KUKA KRL program: ho_axor_atego.src, ho_axor_atego.dat

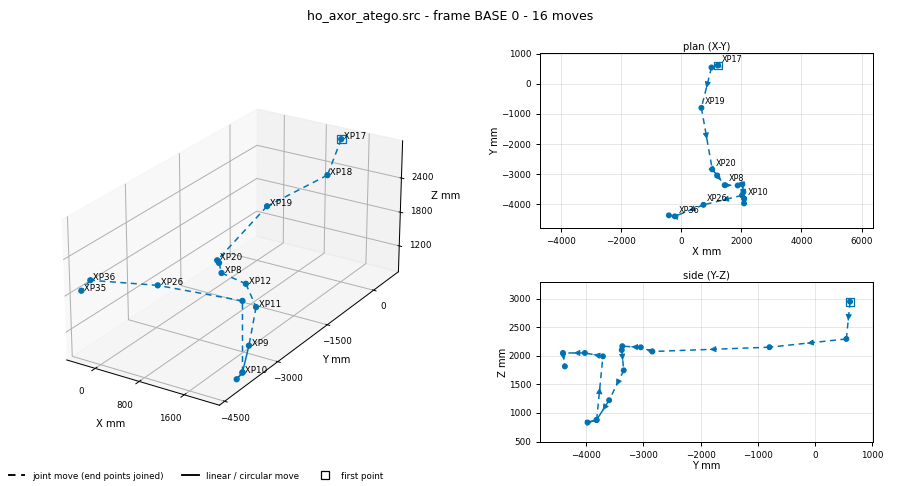
[picture p0: tool path of ho_axor_atego.src in frame BASE 0, 16 of 16 moves have a stored position in this frame; points joined in program order, loops and branches not executed]
--- ho_axor_atego.src ---
&ACCESS RVP
&REL 517
&COMMENT Pega Frente Axor_Atego
&PARAM DISKPATH = KRC:\R1\Program
&PARAM TEMPLATE = C:\KRC\Roboter\Template\vorgabe
&PARAM EDITMASK = *
DEF ho_axor_atego( )
;FOLD INI
  ;FOLD BASISTECH INI
    GLOBAL INTERRUPT DECL 3 WHEN $STOPMESS==TRUE DO IR_STOPM ( )
    INTERRUPT ON 3
    BAS (#INITMOV,0 )
  ;ENDFOLD (BASISTECH INI)
;FOLD SPOTTECH INI
USERSPOT(#INIT)
;ENDFOLD (SPOTTECH INI)
;FOLD GRIPPERTECH INI
USER_GRP(0,DUMMY,DUMMY,GDEFAULT)
;ENDFOLD (GRIPPERTECH INI)
  ;FOLD USER INI
    ;Make your modifications here

  ;ENDFOLD (USER INI)
;ENDFOLD (INI)

; Caracterização dos meios de produção:
; Changes: Pega Frontal Axor/Atego
; Versão Atual:11/08/2015
; Name: P13.050-R4

chk_w6_wechs_ok ( )  ; CHECK TOOL: GRIPPER AXOR

;FOLD PTP P17 Vel=100 % PDAT16 Tool[6]:GARRA AXOR Base[0];%{PE}%R 8.2.20,%MKUKATPBASIS,%CMOVE,%VPTP,%P 1:PTP, 2:P17, 3:, 5:100, 7:PDAT16
$BWDSTART=FALSE
PDAT_ACT=PPDAT16
FDAT_ACT=FP17
BAS(#PTP_PARAMS,100)
PTP XP17
;ENDFOLD

;FOLD PTP P18 CONT Vel=100 % PDAT17 Tool[6]:GARRA AXOR Base[0];%{PE}%R 8.2.20,%MKUKATPBASIS,%CMOVE,%VPTP,%P 1:PTP, 2:P18, 3:C_DIS, 5:100, 7:PDAT17
$BWDSTART=FALSE
PDAT_ACT=PPDAT17
FDAT_ACT=FP18
BAS(#PTP_PARAMS,100)
PTP XP18 C_DIS
;ENDFOLD
;FOLD PTP P19 CONT Vel=100 % PDAT18 Tool[6]:GARRA AXOR Base[0];%{PE}%R 8.2.20,%MKUKATPBASIS,%CMOVE,%VPTP,%P 1:PTP, 2:P19, 3:C_DIS, 5:100, 7:PDAT18
$BWDSTART=FALSE
PDAT_ACT=PPDAT18
FDAT_ACT=FP19
BAS(#PTP_PARAMS,100)
PTP XP19 C_DIS
;ENDFOLD

;FOLD ; LIBERACAO P/ RETIRAR PECA NO DISPOSITIVO;%{PE}%R 8.2.20,%MKUKATPBASIS,%CCOMMENT,%VNORMAL,%P 2:LIBERACAO  P/  RETIRAR  PECA  NO  DISPOSITIVO
;ENDFOLD
;FOLD PTP P20 CONT Vel=100 % PDAT19 Tool[6]:GARRA AXOR Base[0];%{PE}%R 8.2.20,%MKUKATPBASIS,%CMOVE,%VPTP,%P 1:PTP, 2:P20, 3:C_DIS, 5:100, 7:PDAT19
$BWDSTART=FALSE
PDAT_ACT=PPDAT19
FDAT_ACT=FP20
BAS(#PTP_PARAMS,100)
PTP XP20 C_DIS
;ENDFOLD

;FOLD OUT 3352 'R4 busca peca Actros' State=TRUE ;%{PE}%R 8.2.20,%MKUKATPBASIS,%COUT,%VOUTX,%P 2:3352, 3:R4 busca peca Actros, 5:TRUE, 6:
$OUT[3352]=TRUE
;ENDFOLD
;FOLD WAIT FOR ( IN 3352 'Aguarda lib buscar peca Actros' );%{PE}%R 8.2.20,%MKUKATPBASIS,%CEXT_WAIT_FOR,%VEXT_WAIT_FOR,%P 2:, 4:, 5:$IN, 6:3352, 7:Aguarda lib buscar peca Actros, 9:
WAIT FOR  ( $IN[3352] )
;ENDFOLD
;FOLD OUT 3352 'R4 busca peca Actros' State=FALSE ;%{PE}%R 8.2.20,%MKUKATPBASIS,%COUT,%VOUTX,%P 2:3352, 3:R4 busca peca Actros, 5:FALSE, 6:
$OUT[3352]=FALSE
;ENDFOLD
;FOLD OUT 3342 'Fora area externa' State=FALSE ;%{PE}%R 8.2.20,%MKUKATPBASIS,%COUT,%VOUTX,%P 2:3342, 3:Fora area externa, 5:FALSE, 6:
$OUT[3342]=FALSE
;ENDFOLD

;FOLD PTP P15 CONT Vel=100 % PDAT14 Tool[6]:GARRA AXOR Base[0];%{PE}%R 8.2.20,%MKUKATPBASIS,%CMOVE,%VPTP,%P 1:PTP, 2:P15, 3:C_DIS, 5:100, 7:PDAT14
$BWDSTART=FALSE
PDAT_ACT=PPDAT14
FDAT_ACT=FP15
BAS(#PTP_PARAMS,100)
PTP XP15 C_DIS
;ENDFOLD
;FOLD PTP P8 CONT Vel=100 % PDAT9 Tool[6]:GARRA AXOR Base[0];%{PE}%R 8.2.20,%MKUKATPBASIS,%CMOVE,%VPTP,%P 1:PTP, 2:P8, 3:C_DIS, 5:100, 7:PDAT9
$BWDSTART=FALSE
PDAT_ACT=PPDAT9
FDAT_ACT=FP8
BAS(#PTP_PARAMS,100)
PTP XP8 C_DIS
;ENDFOLD
;FOLD PTP P12 CONT Vel=100 % PDAT12 Tool[6]:GARRA AXOR Base[0];%{PE}%R 8.2.20,%MKUKATPBASIS,%CMOVE,%VPTP,%P 1:PTP, 2:P12, 3:C_DIS, 5:100, 7:PDAT12
$BWDSTART=FALSE
PDAT_ACT=PPDAT12
FDAT_ACT=FP12
BAS(#PTP_PARAMS,100)
PTP XP12 C_DIS
;ENDFOLD
;FOLD PTP P11 CONT Vel=100 % PDAT11 Tool[6]:GARRA AXOR Base[0];%{PE}%R 8.2.20,%MKUKATPBASIS,%CMOVE,%VPTP,%P 1:PTP, 2:P11, 3:C_DIS, 5:100, 7:PDAT11
$BWDSTART=FALSE
PDAT_ACT=PPDAT11
FDAT_ACT=FP11
BAS(#PTP_PARAMS,100)
PTP XP11 C_DIS
;ENDFOLD
;FOLD PTP P9 CONT Vel=100 % PDAT10 Tool[6]:GARRA AXOR Base[0];%{PE}%R 8.2.20,%MKUKATPBASIS,%CMOVE,%VPTP,%P 1:PTP, 2:P9, 3:C_DIS, 5:100, 7:PDAT10
$BWDSTART=FALSE
PDAT_ACT=PPDAT10
FDAT_ACT=FP9
BAS(#PTP_PARAMS,100)
PTP XP9 C_DIS
;ENDFOLD

;FOLD SET Z1.1/Z1.2/Z1.3 AXOR State=OPN GDAT12;%{PE}%R 8.2.1,%MKUKATPGRP,%CGRP,%VGRP,%P 2:5, 4:1, 5:#NO, 6:GDAT12, 8:0, 10:0
H50(GRP,5,1,GGDAT12)
;ENDFOLD
;FOLD SET Z2.1/Z2.2 AXOR State=OPN GDAT13;%{PE}%R 8.2.1,%MKUKATPGRP,%CGRP,%VGRP,%P 2:6, 4:1, 5:#NO, 6:GDAT13, 8:0, 10:0
H50(GRP,6,1,GGDAT13)
;ENDFOLD
;FOLD SET Z3.1/Z3.2 AXOR State=OPN GDAT14;%{PE}%R 8.2.1,%MKUKATPGRP,%CGRP,%VGRP,%P 2:7, 4:1, 5:#NO, 6:GDAT14, 8:0, 10:0
H50(GRP,7,1,GGDAT14)
;ENDFOLD
chk_w6_grp1_opn ()
chk_w6_grp2_opn ()
chk_w6_grp3_opn ()

;FOLD LIN P10 CONT Vel=0.5 m/s CPDAT3 Tool[6]:GARRA AXOR Base[0];%{PE}%R 8.2.20,%MKUKATPBASIS,%CMOVE,%VLIN,%P 1:LIN, 2:P10, 3:C_DIS C_DIS, 5:0.5, 7:CPDAT3
$BWDSTART=FALSE
LDAT_ACT=LCPDAT3
FDAT_ACT=FP10
BAS(#CP_PARAMS,0.5)
LIN XP10 C_DIS C_DIS
;ENDFOLD

;FOLD ; POSICAO DE PEGA DA PECA;%{PE}%R 8.2.20,%MKUKATPBASIS,%CCOMMENT,%VNORMAL,%P 2:POSICAO  DE  PEGA  DA  PECA
;ENDFOLD
;FOLD LIN P14 CONT Vel=0.5 m/s CPDAT4 Tool[6]:GARRA AXOR Base[0];%{PE}%R 8.2.20,%MKUKATPBASIS,%CMOVE,%VLIN,%P 1:LIN, 2:P14, 3:C_DIS C_DIS, 5:0.5, 7:CPDAT4
$BWDSTART=FALSE
LDAT_ACT=LCPDAT4
FDAT_ACT=FP14
BAS(#CP_PARAMS,0.5)
LIN XP14 C_DIS C_DIS
;ENDFOLD

IF (NOT(GHOST())) THEN
;FOLD WAIT FOR ( IN 489 'Presença de peça 1 - Axor' AND IN 490 'Presença de peça 2 - Axor' );%{PE}%R 8.2.20,%MKUKATPBASIS,%CEXT_WAIT_FOR,%VEXT_WAIT_FOR,%P 2:, 4:, 5:$IN, 6:489, 7:Presença de peça 1 - Axor, 8:AND, 9:, 10:$IN, 11:490, 12:Presença de peça 2 - Axor, 14:
WAIT FOR  ( $IN[489] AND $IN[490] )
;ENDFOLD
ENDIF

;FOLD SET Z1.1/Z1.2/Z1.3 AXOR State=CLO GDAT9;%{PE}%R 8.2.1,%MKUKATPGRP,%CGRP,%VGRP,%P 2:5, 4:2, 5:#NO, 6:GDAT9, 8:0, 10:0
H50(GRP,5,2,GGDAT9)
;ENDFOLD
;FOLD SET Z2.1/Z2.2 AXOR State=CLO GDAT10;%{PE}%R 8.2.1,%MKUKATPGRP,%CGRP,%VGRP,%P 2:6, 4:2, 5:#NO, 6:GDAT10, 8:0, 10:0
H50(GRP,6,2,GGDAT10)
;ENDFOLD
;FOLD SET Z3.1/Z3.2 AXOR State=CLO GDAT11;%{PE}%R 8.2.1,%MKUKATPGRP,%CGRP,%VGRP,%P 2:7, 4:2, 5:#NO, 6:GDAT11, 8:0, 10:0
H50(GRP,7,2,GGDAT11)
;ENDFOLD
chk_w6_grp1_clo ()
chk_w6_grp2_clo ()
chk_w6_grp3_clo ()

;FOLD OUT 3349 'R4 pegou peca' State=TRUE ;%{PE}%R 8.2.20,%MKUKATPBASIS,%COUT,%VOUTX,%P 2:3349, 3:R4 pegou peca, 5:TRUE, 6:
$OUT[3349]=TRUE
;ENDFOLD
;FOLD OUT 3350 'R4 solicita lib sair magazine' State=TRUE ;%{PE}%R 8.2.20,%MKUKATPBASIS,%COUT,%VOUTX,%P 2:3350, 3:R4 solicita lib sair magazine, 5:TRUE, 6:
$OUT[3350]=TRUE
;ENDFOLD
;FOLD WAIT FOR ( IN 3349 'Aguarda lib sair magazine' );%{PE}%R 8.2.20,%MKUKATPBASIS,%CEXT_WAIT_FOR,%VEXT_WAIT_FOR,%P 2:, 4:, 5:$IN, 6:3349, 7:Aguarda lib sair magazine, 9:
WAIT FOR  ( $IN[3349] )
;ENDFOLD
;FOLD OUT 3350 'R4 solicita lib sair magazine' State=FALSE ;%{PE}%R 8.2.20,%MKUKATPBASIS,%COUT,%VOUTX,%P 2:3350, 3:R4 solicita lib sair magazine, 5:FALSE, 6:
$OUT[3350]=FALSE
;ENDFOLD

;FOLD LIN P22 CONT Vel=0.1 m/s CPDAT6 Tool[6]:GARRA AXOR Base[0];%{PE}%R 8.2.20,%MKUKATPBASIS,%CMOVE,%VLIN,%P 1:LIN, 2:P22, 3:C_DIS C_DIS, 5:0.1, 7:CPDAT6
$BWDSTART=FALSE
LDAT_ACT=LCPDAT6
FDAT_ACT=FP22
BAS(#CP_PARAMS,0.1)
LIN XP22 C_DIS C_DIS
;ENDFOLD

IF (NOT(GHOST())) THEN
;FOLD WAIT FOR ( IN 489 'Presença de peça 1 - Axor' AND IN 490 'Presença de peça 2 - Axor' );%{PE}%R 8.2.20,%MKUKATPBASIS,%CEXT_WAIT_FOR,%VEXT_WAIT_FOR,%P 2:, 4:, 5:$IN, 6:489, 7:Presença de peça 1 - Axor, 8:AND, 9:, 10:$IN, 11:490, 12:Presença de peça 2 - Axor, 14:
WAIT FOR  ( $IN[489] AND $IN[490] )
;ENDFOLD
ENDIF

;FOLD PTP P25 CONT Vel=100 % PDAT23 Tool[6]:GARRA AXOR Base[0];%{PE}%R 8.2.20,%MKUKATPBASIS,%CMOVE,%VPTP,%P 1:PTP, 2:P25, 3:C_DIS, 5:100, 7:PDAT23
$BWDSTART=FALSE
PDAT_ACT=PPDAT23
FDAT_ACT=FP25
BAS(#PTP_PARAMS,100)
PTP XP25 C_DIS
;ENDFOLD
;FOLD PTP P26 CONT Vel=100 % PDAT24 Tool[6]:GARRA AXOR Base[0];%{PE}%R 8.2.20,%MKUKATPBASIS,%CMOVE,%VPTP,%P 1:PTP, 2:P26, 3:C_DIS, 5:100, 7:PDAT24
$BWDSTART=FALSE
PDAT_ACT=PPDAT24
FDAT_ACT=FP26
BAS(#PTP_PARAMS,100)
PTP XP26 C_DIS
;ENDFOLD
;FOLD PTP P36 CONT Vel=100 % PDAT33 Tool[6]:GARRA AXOR Base[0];%{PE}%R 8.2.20,%MKUKATPBASIS,%CMOVE,%VPTP,%P 1:PTP, 2:P36, 3:C_DIS, 5:100, 7:PDAT33
$BWDSTART=FALSE
PDAT_ACT=PPDAT33
FDAT_ACT=FP36
BAS(#PTP_PARAMS,100)
PTP XP36 C_DIS
;ENDFOLD
;FOLD PTP P35 CONT Vel=100 % PDAT32 Tool[6]:GARRA AXOR Base[0];%{PE}%R 8.2.20,%MKUKATPBASIS,%CMOVE,%VPTP,%P 1:PTP, 2:P35, 3:C_DIS, 5:100, 7:PDAT32
$BWDSTART=FALSE
PDAT_ACT=PPDAT32
FDAT_ACT=FP35
BAS(#PTP_PARAMS,100)
PTP XP35 C_DIS
;ENDFOLD

END

--- ho_axor_atego.dat ---
&ACCESS RVP
&REL 517
&COMMENT Pega Frente Axor_Atego
&PARAM DISKPATH = KRC:\R1\Program
&PARAM TEMPLATE = C:\KRC\Roboter\Template\vorgabe
&PARAM EDITMASK = *
DEFDAT  ho_axor_atego
;FOLD EXTERNAL DECLARATIONS;%{PE}%MKUKATPBASIS,%CEXT,%VCOMMON,%P
;FOLD GRIPPERTECH EXT
EXT  H50 (INT  :IN,INT  :IN,INT  :IN,GRP_TYP  :IN )
;ENDFOLD (GRIPPERTECH EXT)
;FOLD SPOTTECH EXT
EXT  USERSPOT (S_COMMAND  :IN,SPOT_TYPE  :IN )
;ENDFOLD (SPOTTECH EXT)
;FOLD BASISTECH EXT;%{PE}%MKUKATPBASIS,%CEXT,%VEXT,%P
EXT  BAS (BAS_COMMAND  :IN,REAL  :IN )
DECL INT SUCCESS
;ENDFOLD (BASISTECH EXT)
;FOLD USER EXT;%{E}%MKUKATPUSER,%CEXT,%VEXT,%P
;Make your modifications here

;ENDFOLD (USER EXT)
;ENDFOLD (EXTERNAL DECLARATIONS)
DECL BASIS_SUGG_T LAST_BASIS={POINT1[] "P37                     ",POINT2[] "P37                     ",CP_PARAMS[] "CPDAT7                  ",PTP_PARAMS[] "PDAT34                  ",CONT[] "C_DIS                   ",CP_VEL[] "0.1                     ",PTP_VEL[] "100                     ",SYNC_PARAMS[] "SYNCDAT                 ",SPL_NAME[] "S0                      "}
DECL E6POS XP8={X 1445.68298,Y -3370.3269,Z 2167.86108,A -26.0050793,B 77.6218033,C -0.625826001,S 2,T 35,E1 3350.18604,E2 0.0,E3 0.0,E4 0.0,E5 0.0,E6 0.0}
DECL FDAT FP8={TOOL_NO 6,BASE_NO 0,IPO_FRAME #BASE,POINT2[] " ",TQ_STATE FALSE}
DECL E6POS XP9={X 2069.63599,Y -3600.41699,Z 1223.01794,A 73.2965622,B 80.4088898,C 148.646393,S 2,T 35,E1 2952.2561,E2 0.0,E3 0.0,E4 0.0,E5 0.0,E6 0.0}
DECL FDAT FP9={TOOL_NO 6,BASE_NO 0,IPO_FRAME #BASE,POINT2[] " ",TQ_STATE FALSE}
DECL E6POS XP10={X 2093.60791,Y -3821.00391,Z 876.983887,A 88.6464615,B 74.6173401,C 179.506302,S 2,T 35,E1 2929.21606,E2 0.0,E3 0.0,E4 0.0,E5 0.0,E6 0.0}
DECL FDAT FP10={TOOL_NO 6,BASE_NO 0,IPO_FRAME #BASE,POINT2[] " ",TQ_STATE FALSE}
DECL LDAT LCPDAT3={VEL 2.0,ACC 100.0,APO_DIST 100.0,APO_FAC 50.0,AXIS_VEL 100.0,AXIS_ACC 100.0,ORI_TYP #VAR,CIRC_TYP #BASE,JERK_FAC 50.0,GEAR_JERK 50.0,EXAX_IGN 0}
DECL PDAT PPDAT9={VEL 100.0,ACC 100.0,APO_DIST 100.0,APO_MODE #CDIS}
DECL PDAT PPDAT10={VEL 100.0,ACC 100.0,APO_DIST 100.0,APO_MODE #CDIS}
DECL E6POS XP11={X 2035.30298,Y -3345.36401,Z 1745.60901,A 2.13454509,B 83.8452072,C 54.8674812,S 2,T 35,E1 2985.87988,E2 0.0,E3 0.0,E4 0.0,E5 0.0,E6 0.0}
DECL FDAT FP11={TOOL_NO 6,BASE_NO 0,IPO_FRAME #BASE,POINT2[] " ",TQ_STATE FALSE}
DECL PDAT PPDAT11={VEL 100.0,ACC 100.0,APO_DIST 100.0,APO_MODE #CDIS}
DECL E6POS XP12={X 1878.09998,Y -3379.83911,Z 2101.00903,A -35.0093994,B 79.7438202,C 2.34273291,S 2,T 35,E1 3008.74707,E2 0.0,E3 0.0,E4 0.0,E5 0.0,E6 0.0}
DECL FDAT FP12={TOOL_NO 6,BASE_NO 0,IPO_FRAME #BASE,POINT2[] " ",TQ_STATE FALSE}
DECL PDAT PPDAT12={VEL 100.0,ACC 100.0,APO_DIST 100.0,APO_MODE #CDIS}
DECL E6POS XP14={X 2091.30591,Y -3977.78198,Z 833.848022,A 88.6464615,B 74.6173401,C 179.506302,S 2,T 35,E1 2929.21606,E2 0.0,E3 0.0,E4 0.0,E5 0.0,E6 0.0}
DECL FDAT FP14={TOOL_NO 6,BASE_NO 0,IPO_FRAME #BASE,POINT2[] " ",TQ_STATE FALSE}
DECL LDAT LCPDAT4={VEL 2.0,ACC 100.0,APO_DIST 100.0,APO_FAC 50.0,AXIS_VEL 100.0,AXIS_ACC 100.0,ORI_TYP #VAR,CIRC_TYP #BASE,JERK_FAC 50.0,GEAR_JERK 50.0,EXAX_IGN 0}
DECL E6POS XP15={X 1194.80603,Y -3046.59912,Z 2147.95605,A -7.891541,B 84.4729614,C 1.08770204,S 2,T 35,E1 3350.18701,E2 0.0,E3 0.0,E4 0.0,E5 0.0,E6 0.0}
DECL FDAT FP15={TOOL_NO 6,BASE_NO 0,IPO_FRAME #BASE,POINT2[] " ",TQ_STATE FALSE}
DECL PDAT PPDAT14={VEL 100.0,ACC 100.0,APO_DIST 100.0,APO_MODE #CDIS}
DECL PDAT PPDAT16={VEL 100.0,ACC 100.0,APO_DIST 100.0,APO_MODE #CDIS}
DECL E6POS XP17={X 1215.88794,Y 611.95752,Z 2946.29297,A -37.8803101,B 80.3210068,C -65.6440201,S 2,T 35,E1 -86.9784317,E2 0.0,E3 0.0,E4 0.0,E5 0.0,E6 0.0}
DECL FDAT FP17={TOOL_NO 6,BASE_NO 0,IPO_FRAME #BASE,POINT2[] " ",TQ_STATE FALSE}
DECL PDAT PPDAT17={VEL 100.0,ACC 100.0,APO_DIST 100.0,APO_MODE #CDIS}
DECL E6POS XP18={X 1006.51001,Y 547.768494,Z 2294.32104,A 25.3571892,B 87.6897507,C 20.4661694,S 2,T 35,E1 -86.978302,E2 0.0,E3 0.0,E4 0.0,E5 0.0,E6 0.0}
DECL FDAT FP18={TOOL_NO 6,BASE_NO 0,IPO_FRAME #BASE,POINT2[] " ",TQ_STATE FALSE}
DECL PDAT PPDAT18={VEL 100.0,ACC 100.0,APO_DIST 100.0,APO_MODE #CDIS}
DECL E6POS XP19={X 671.108582,Y -796.590271,Z 2150.08398,A 33.6693993,B 82.7202377,C 2.89461398,S 2,T 35,E1 1710.36499,E2 0.0,E3 0.0,E4 0.0,E5 0.0,E6 0.0}
DECL FDAT FP19={TOOL_NO 6,BASE_NO 0,IPO_FRAME #BASE,POINT2[] " ",TQ_STATE FALSE}
DECL PDAT PPDAT19={VEL 100.0,ACC 100.0,APO_DIST 100.0,APO_MODE #CDIS}
DECL E6POS XP20={X 1033.07703,Y -2844.12793,Z 2074.83008,A 4.45546293,B 89.221138,C 2.08266401,S 2,T 35,E1 3350.18701,E2 0.0,E3 0.0,E4 0.0,E5 0.0,E6 0.0}
DECL FDAT FP20={TOOL_NO 6,BASE_NO 0,IPO_FRAME #BASE,POINT2[] " ",TQ_STATE FALSE}
DECL GRP_SUGG_T LAST_GRP={NUMBER[] "7                       ",STATE[] "2                       ",PARAMS[] "GDAT11                  "}
DECL GRP_TYP GGDAT2={G_APO #NO,GRP_TIME 0.200000003,CTRL #OFF,DLY 0,DST 1}
DECL GRP_TYP GGDAT3={G_APO #NO,GRP_TIME 0.200000003,CTRL #OFF,DLY 0,DST 1}
DECL GRP_TYP GGDAT4={G_APO #NO,GRP_TIME 0.200000003,CTRL #OFF,DLY 0,DST 1}
DECL GRP_TYP GGDAT5={G_APO #NO,GRP_TIME 0.200000003,CTRL #OFF,DLY 0,DST 1}
DECL GRP_TYP GGDAT1={G_APO #NO,GRP_TIME 0.200000003,CTRL #OFF,DLY 0,DST 1}
DECL GRP_TYP GGDAT6={G_APO #NO,GRP_TIME 0.200000003,CTRL #OFF,DLY 0,DST 1}
DECL GRP_TYP GGDAT7={G_APO #NO,GRP_TIME 0.200000003,CTRL #OFF,DLY 0,DST 1}
DECL GRP_TYP GGDAT8={G_APO #NO,GRP_TIME 0.200000003,CTRL #OFF,DLY 0,DST 1}
DECL E6POS XP22={X 2093.63892,Y -3818.90601,Z 877.546387,A 88.6445007,B 74.617157,C 179.504593,S 2,T 35,E1 2929.21704,E2 0.0,E3 0.0,E4 0.0,E5 0.0,E6 0.0}
DECL FDAT FP22={TOOL_NO 7,BASE_NO 0,IPO_FRAME #BASE,POINT2[] " ",TQ_STATE FALSE}
DECL LDAT LCPDAT6={VEL 2.0,ACC 100.0,APO_DIST 100.0,APO_FAC 50.0,AXIS_VEL 100.0,AXIS_ACC 100.0,ORI_TYP #VAR,CIRC_TYP #BASE,JERK_FAC 50.0,GEAR_JERK 50.0,EXAX_IGN 0}
DECL GRP_TYP GGDAT9={G_APO #NO,GRP_TIME 0.200000003,CTRL #OFF,DLY 0,DST 1}
DECL GRP_TYP GGDAT10={G_APO #NO,GRP_TIME 0.200000003,CTRL #OFF,DLY 0,DST 1}
DECL GRP_TYP GGDAT11={G_APO #NO,GRP_TIME 0.200000003,CTRL #OFF,DLY 0,DST 1}
DECL GRP_TYP GCONT={G_APO #YES,GRP_TIME 0.0,CTRL #OFF,DLY 0,DST 0}
DECL E6POS XP25={X 2023.86804,Y -3709.19092,Z 1990.57495,A -122.206497,B 81.4805984,C -46.6409683,S 2,T 35,E1 2368.08008,E2 0.0,E3 0.0,E4 0.0,E5 0.0,E6 0.0}
DECL FDAT FP25={TOOL_NO 7,BASE_NO 0,IPO_FRAME #BASE,POINT2[] " ",TQ_STATE FALSE}
DECL PDAT PPDAT23={VEL 100.0,ACC 100.0,APO_DIST 100.0,APO_MODE #CDIS}
DECL E6POS XP26={X 739.380981,Y -4024.96997,Z 2049.55591,A -73.0736237,B 82.7862625,C -2.68507004,S 2,T 35,E1 2134.42896,E2 0.0,E3 0.0,E4 0.0,E5 0.0,E6 0.0}
DECL FDAT FP26={TOOL_NO 7,BASE_NO 0,IPO_FRAME #BASE,POINT2[] " ",TQ_STATE FALSE}
DECL PDAT PPDAT24={VEL 100.0,ACC 100.0,APO_DIST 100.0,APO_MODE #CDIS}
DECL GRP_TYP GGDAT12={G_APO #NO,GRP_TIME 0.200000003,CTRL #OFF,DLY 0,DST 1}
DECL GRP_TYP GGDAT13={G_APO #NO,GRP_TIME 0.200000003,CTRL #OFF,DLY 0,DST 1}
DECL GRP_TYP GGDAT14={G_APO #NO,GRP_TIME 0.200000003,CTRL #OFF,DLY 0,DST 1}
DECL E6POS XP35={X -411.517609,Y -4374.29785,Z 1814.03601,A -89.77034,B 87.6975327,C -41.8600388,S 2,T 34,E1 2400.13794,E2 0.0,E3 0.0,E4 0.0,E5 0.0,E6 0.0}
DECL FDAT FP35={TOOL_NO 7,BASE_NO 0,IPO_FRAME #BASE,POINT2[] " ",TQ_STATE FALSE}
DECL PDAT PPDAT32={VEL 100.0,ACC 100.0,APO_DIST 100.0,APO_MODE #CDIS}
DECL E6POS XP36={X -213.805298,Y -4407.87305,Z 2049.55298,A -73.0732727,B 82.7863083,C -2.68476701,S 2,T 34,E1 2134.42993,E2 0.0,E3 0.0,E4 0.0,E5 0.0,E6 0.0}
DECL FDAT FP36={TOOL_NO 7,BASE_NO 0,IPO_FRAME #BASE,POINT2[] " ",TQ_STATE FALSE}
DECL PDAT PPDAT33={VEL 100.0,ACC 100.0,APO_DIST 100.0,APO_MODE #CDIS}
ENDDAT
